(* IEC 61131-3 sources: iec-checker/test/st, 29 files *)

(* ---- declaration-analysis.st ---- *)
(* This demo includes some declaration errors *)
TYPE
    (* String types *)
    ST0 : STRING[5];                               (* OK *)
    ST1 : STRING;                                  (* OK *)
    ST2 : STRING[5] := 'foo';                      (* OK *)
    ST3 : STRING := 'platform_dependent';          (* OK *)
    ST4 : STRING[5] := "foobar";                   (* Error *)

    (* Subrange types *)
    ANALOG_DATA1 : INT (-4095 .. 4095);          (* OK *)
    ANALOG_DATA1 : INT (-4095 .. 4095) := 2000;  (* OK *)
    ANALOG_DATA1 : INT (-4095 .. 4095) := 4095;  (* OK: See 6.4.4.4.1 *)
    ANALOG_DATA1 : INT (-4095 .. 4095) := -4095; (* OK: See 6.4.4.4.1 *)
    ANALOG_DATA2 : INT (-4095 .. 4095) := 4099;  (* Error *)
    ANALOG_DATA2 : INT (-4095 .. 4095) := -4096; (* Error *)
END_TYPE

(* ---- merge-1.st ---- *)
TYPE example_struct :
  STRUCT
    Field : BOOL;
  END_STRUCT
END_TYPE

(* ---- plcopen-cp13.st ---- *)
(* Uncompatible: Recursive functions are forbidden *)
FUNCTION Factorial : INT
    VAR_INPUT
        X : INT;
    END_VAR

    IF X > 1 THEN
        Factorial := Factorial(X - 1) * X;
    ELSE
        Factorial := X;
    END_IF;
END_FUNCTION

(* Compatible iterative implementation *)
FUNCTION Factorial_good : INT
    VAR_INPUT
        X : INT;
    END_VAR
    VAR
        Acc : INT;
    END_VAR

    FOR I := 0 TO 100 DO
        Acc := Acc * X;
    END_FOR;
    Factorial := Acc;
END_FUNCTION

(* ---- plcopen-cp3.st ---- *)
FUNCTION demo : INT
    VAR_INPUT
        x1 : INT := 0;
        x2 : INT; (* PLCOPEN-CP3 *)
        x3 : STRING[5]; (* PLCOPEN-CP3 *)
        x4 : WSTRING[25] := 'spaces_disallowed';
        x5 : ARRAY [1..2, 1..3] OF INT; (* PLCOPEN-CP3 *)
        x6: ARRAY [0..7] OF BOOL := [0,1,1,0,0,1,0,0];
        x7 AT %B0 : INT;
    END_VAR
    x1 := 42;
END_FUNCTION

(* ---- plcopen-cp4.st ---- *)
FUNCTION demo : INT
    VAR_INPUT
        x1 AT %MX40 : INT; (* PLCOPEN-CP4 *)
        x2 AT %MX41 : INT; (* PLCOPEN-CP4 *)
        x3 AT %MX510 : INT;
    END_VAR
    x1 := 42;
END_FUNCTION

(* ---- plcopen-n4.st ---- *)
FUNCTION StartMotor : BOOL
  VAR
    goodVar : INT;
    BadVar  : INT;  (* PLCOPEN-N4 *)
  END_VAR
  StartMotor := TRUE;
END_FUNCTION

FUNCTION start_motor : BOOL    (* PLCOPEN-N4 *)
  start_motor := FALSE;
END_FUNCTION

(* ---- plcopen-n6.st ---- *)
FUNCTION Go : BOOL   (* PLCOPEN-N6 *)
  Go := TRUE;
END_FUNCTION

FUNCTION ReadAndScaleTheTemperatureInput : REAL   (* PLCOPEN-N6 *)
  ReadAndScaleTheTemperatureInput := 0.0;
END_FUNCTION

FUNCTION StartFeeding : BOOL
  StartFeeding := TRUE;
END_FUNCTION

(* ---- plcopen-cp16.st ---- *)
FUNCTION_BLOCK MyFB
  VAR x : INT; END_VAR
  x := 0;
END_FUNCTION_BLOCK

PROGRAM MyProgram
  VAR y : INT; END_VAR
  y := 0;
END_PROGRAM

CONFIGURATION config
  RESOURCE res1 ON PLC
    TASK Fast(INTERVAL := T#10ms, PRIORITY := 1);
    TASK Slow(INTERVAL := T#100ms, PRIORITY := 2);
    PROGRAM inst1 WITH Fast : MyProgram;
    PROGRAM inst2 WITH Slow : MyFB;
    PROGRAM inst3 : MyProgram;
  END_RESOURCE
END_CONFIGURATION

(* ---- plcopen-cp17.st ---- *)
FUNCTION_BLOCK FB_CP17_Test
VAR_INPUT
    in_ok_read_only       : INT;   // Compliant: read at least once, never written
    in_violate_unused     : INT;   // Violation: never read
    in_violate_write_only : INT;   // Violation: written, not read
    in_violate_read_write : INT;   // Violation: read but also written

    idx_read_only           : INT;   // Compliant: only read as array index
    idx_violate_write_only  : INT;   // Violation: written, not read
    func_violate_unused     : INT;   // Violation: never use
    func_read_only          : INT;   // Compliant: only read in func call
    func_violate_write      : INT;   // Violation: written in func call
END_VAR

VAR_OUTPUT
    out_ok_written        : INT;   // Compliant: written at least once
    out_violate_unused    : INT;   // Violation: never written
    out_violate_read_only : INT;   // Violation: read but not written
END_VAR

VAR_IN_OUT
    io_ok_read_only       : INT;   // Compliant: read only
    io_ok_write_only      : INT;   // Compliant: written only
    io_ok_read_write      : INT;   // Compliant: both read and written
    io_violate_unused     : INT;   // Violation: neither read nor written
END_VAR

VAR
    temp : INT;
    arr  : ARRAY[0..9] OF INT;
    func : MYFUNC;
END_VAR

(* ===== VAR_INPUT tests ===== *)

(* Compliant: input parameter is read *)
temp := in_ok_read_only + 1;

(* Violation: in_violate_unused is never used *)

(* Violation: input parameter is written *)
in_violate_write_only := 100;

(* Violation: input parameter is both read and written *)
temp := in_violate_read_write;
in_violate_read_write := temp + 1;

(* ===== VAR_OUTPUT tests ===== *)

(* Compliant: output parameter is written *)
out_ok_written := temp;

(* Violation: out_violate_unused is never written *)

(* Violation: output parameter is read but not written *)
temp := out_violate_read_only;

(* ===== VAR_IN_OUT tests ===== *)

(* Compliant: read only *)
temp := temp + io_ok_read_only;

(* Compliant: written only *)
io_ok_write_only := 10;

(* Compliant: both read and written *)
io_ok_read_write := io_ok_read_write + 1;

(* Violation: io_violate_unused is never used *)

(* ===== special tests for LHS handling ===== *)

(* Important case:
   idx_read_only is used only to locate the write target arr[idx_read_only].
   It should be counted as READ, not WRITE.
   However, *)
arr[idx_read_only] := 5;

(* Violation:
   idx_violate_write_only is written, but never read. *)
idx_violate_write_only := 3;

(* Function Call *)
func(func_violate_unused := func_read_only, func_violate_unused => func_violate_write);

END_FUNCTION_BLOCK

(*
 * The reported result should be:
 * 1. in_violate_unused => should be read
 * 2. in_violate_write_only => should not be written, should be read (2 * warnings reported)
 * 3. in_violate_read_write => should not be written
 * 4. out_violate_unused => should be written
 * 5. out_violate_read_only => should be written
 * 6. io_violate_unused => should be written/read
 * 7. idx_violate_write_only => should not be written, should be read (2 * warnings reported)
 * 8. func_violate_unused => never used, should be read
 * 9. func_violate_write => should not be written, should be read (2 * warnings reported)
*)

(* ---- plcopen-cp6.st ---- *)
FUNCTION demo : INT
    VAR_EXTERNAL
        x1 : INT; (* PLCOPEN-CP6 *)
    END_VAR
    x1 := 42;
END_FUNCTION

FUNCTION_BLOCK demo
    VAR_EXTERNAL
        x1 : INT; (* PLCOPEN-CP6 *)
    END_VAR
    x1 := 42;
END_FUNCTION_BLOCK

PROGRAM demo
    VAR_EXTERNAL
        x1 : INT;
    END_VAR
    x1 := 42;
END_PROGRAM

CLASS test1
  VAR_EXTERNAL
    x1 : INT;
  END_VAR

  METHOD PRIVATE count
    x1 := 42;
  END_METHOD

END_CLASS

(* ---- plcopen-cp9.st ---- *)
(* Example from PLCOpen guidelines, page 60.

   The following Function block CHARCURVE has:
   Number of Statements 18
   McCabe complexity of 12
   Prater complexity of 3,89
   Halstead complexity of 44,9
   Elshof complexity of 0,14

  NOTE: I'm not sure how they evaluated number of statements and appropriate
  complexity metrics. I have 4 additional statements for this program, and it
  seems correct for me.
 *)

FUNCTION_BLOCK CHARCURVE
  VAR_INPUT
    IN:INT;
    N:BYTE;
  END_VAR
  (* VAR_IN_OUT *)
    (* P : ARRAY [0 .. 10] OF POINT; *)
  (* END_VAR *)
  VAR_OUTPUT
    OUT:INT;
    ERR: BYTE;
  END_VAR
  VAR
    I:INT;
  END_VAR

  IF N > 1 AND N < 12 THEN
    ERR:=0;
    (* IF IN < P[0].X THEN *)
    IF IN < a THEN
      ERR := 2;
      OUT := DINT_TO_INT(a);
    (* ELSIF IN > P[N-1].X THEN *)
    ELSIF IN > a THEN
      ERR := 2;
      OUT := DINT_TO_INT(a);
    ELSE
      FOR I:=1 TO N-1 DO
        (* IF P[I-1].X >= P[I].X THEN *)
        IF a >= a THEN
          ERR:=1;
          EXIT;
        END_IF;
        (* IF IN <= P[I].X THEN *)
        IF IN <= a THEN
          EXIT;
        END_IF;
      END_FOR;
      IF ERR = 0 THEN
        (* OUT := DINT_TO_INT(P[I].Y - (P[I].X-IN) * (P[I].Y-P[I-1].Y) / (P[I].X-P[I-1].X)); *)
        OUT := DINT_TO_INT(a - (a - IN) * (a - a) / (a - a));
      ELSE
        OUT:=0;
      END_IF;
    END_IF;
  ELSE
    ERR := 4;
  END_IF;
END_FUNCTION_BLOCK

(* ---- plcopen-n10.st ---- *)
TYPE
  Color : (Red, Green, Blue);   (* PLCOPEN-N10 *)
END_TYPE

TYPE
  E_Direction : (North, South, East, West);
END_TYPE

FUNCTION_BLOCK Motor   (* PLCOPEN-N10 *)
  VAR
    speed : INT;
  END_VAR
  speed := 0;
END_FUNCTION_BLOCK

FUNCTION_BLOCK FB_Pump
  VAR
    flow : REAL;
  END_VAR
  flow := 0.0;
END_FUNCTION_BLOCK

(* ---- plcopen-n5.st ---- *)
PROGRAM prog0
  VAR
    local0 : INT;
  END_VAR
  local0 := 0;
END_PROGRAM

FUNCTION_BLOCK Example
  VAR
    MyCalculation : REAL;   (* PLCOPEN-N5 *)
  END_VAR
  MyCalculation := 0.0;
END_FUNCTION_BLOCK

CONFIGURATION config
  VAR_GLOBAL
    MyCalculation : REAL;
  END_VAR
  TASK task0(INTERVAL := T#20ms, PRIORITY := 0);
  PROGRAM instance0 WITH task0 : prog0;
END_CONFIGURATION

(* ---- plcopen-n9.st ---- *)
PROGRAM prog0
  VAR
    local0 : INT;
  END_VAR
  local0 := 0;
END_PROGRAM

FUNCTION_BLOCK MyCalculation   (* PLCOPEN-N9 *)
  VAR
    value : REAL;
  END_VAR
  value := 0.0;
END_FUNCTION_BLOCK

CONFIGURATION config
  VAR_GLOBAL
    MyCalculation : REAL;   (* PLCOPEN-N9 *)
  END_VAR
  TASK task0(INTERVAL := T#20ms, PRIORITY := 0);
  PROGRAM instance0 WITH task0 : prog0;
END_CONFIGURATION

(* ---- dead-code.st ---- *)
FUNCTION dead_code_after_return : INT
  VAR
    counter : INT := 0;
    some_var : INT;
  END_VAR
  counter := counter + 1;
  counter := 2 + 2;
  RETURN;
  some_var := SQRT(16#42); (* UnreachableCode error *)
  some_var := 16#42; (* No additional warnings *)
  some_var := 19;
END_FUNCTION

PROGRAM dead_code_in_the_loops
VAR a : INT; i : INT; END_VAR
  WHILE i < 10 DO
    IF i = 5 THEN
      i := i + 1;
      EXIT;
      i := 19; (* UnreachableCode error *)
      i := 42; (* No additional warnings *)
      i := 42;
    ELSIF i = 6 THEN
      CONTINUE;
      i := 3; (* UnreachableCode error *)
      i := 44; (* No additional warnings *)
      i := 19;
    END_IF;
    i := i + 2;
  END_WHILE;
  I := 0;
END_PROGRAM

(* ---- merge-2.st ---- *)
PROGRAM Program1
  VAR
    instance AT %MW500 : example_struct;
  END_VAR

  %MW500 := TRUE;
END_PROGRAM

(* ---- plcopen-cp1.st ---- *)
(** PLCOPEN-CP1 – Access to a member shall be by name *)

PROGRAM program0
  VAR
    head AT %B0 : INT;
  END_VAR
  %B0 := 42;
END_PROGRAM

(* ---- plcopen-cp25.st ---- *)
PROGRAM demo
    VAR
        I : INT := 10;
        J : REAL := 0.55;
    END_VAR

  I := J; (* PLCOPEN-CP25 *)
  J := I; (* PLCOPEN-CP25 *)
  I := REAL_TO_INT(J);
  J := INT_TO_REAL(I);
END_PROGRAM

(* ---- plcopen-cp26.st ---- *)
CONFIGURATION config
  VAR_GLOBAL
    SharedCounter : INT;
    ReadOnlyVar : INT;
    MultiWriter : INT;
  END_VAR
  TASK task0(INTERVAL := T#20ms, PRIORITY := 0);
  PROGRAM instance0 WITH task0 : Program1;
END_CONFIGURATION

(* Case 1: SharedCounter written by Program1 and Program2 — violation in Program2 *)
PROGRAM Program1
  VAR_EXTERNAL SharedCounter : INT; END_VAR
  VAR_EXTERNAL ReadOnlyVar : INT; END_VAR
  VAR x : INT; END_VAR
  SharedCounter := SharedCounter + 1;
  x := ReadOnlyVar;
END_PROGRAM

PROGRAM Program2
  VAR_EXTERNAL SharedCounter : INT; END_VAR
  VAR_EXTERNAL ReadOnlyVar : INT; END_VAR
  VAR x : INT; END_VAR
  SharedCounter := 0;
  x := ReadOnlyVar;
END_PROGRAM

(* Case 2: MultiWriter written by Program3 and Program4 — violation in Program4 *)
PROGRAM Program3
  VAR_EXTERNAL MultiWriter : INT; END_VAR
  MultiWriter := 1;
END_PROGRAM

PROGRAM Program4
  VAR_EXTERNAL MultiWriter : INT; END_VAR
  MultiWriter := 2;
END_PROGRAM

(* ---- plcopen-cp28.st ---- *)
PROGRAM demo
    VAR
        x : TIME;
    END_VAR

    IF x = T#100MS THEN (* PLCOPEN CP-28 *)
      x := x + 1;
    END_IF;

    IF x <> T#100MS THEN (* PLCOPEN CP-28 *)
      x := x + 1;
    END_IF;

    IF T#100MS = x THEN (* PLCOPEN CP-28 *)
      x := x + 1;
    END_IF;

    IF T#100MS <> x THEN (* PLCOPEN CP-28 *)
      x := x + 1;
    END_IF;

    IF REAL_TO_INT(x) <> 0 THEN
      x := x + 1;
    END_IF;
END_PROGRAM

(* ---- plcopen-cp8.st ---- *)
PROGRAM demo
    VAR
        x : REAL;
    END_VAR

    IF x = 0.0 THEN (* PLCOPEN CP-8 *)
      x := x + 1;
    END_IF;

    IF x <> 0.0 THEN (* PLCOPEN CP-8 *)
      x := x + 1;
    END_IF;

    IF 0.0 = x THEN (* PLCOPEN CP-8 *)
      x := x + 1;
    END_IF;

    IF 0.0 <> x THEN (* PLCOPEN CP-8 *)
      x := x + 1;
    END_IF;

    IF REAL_TO_INT(x) <> 0 THEN
      x := x + 1;
    END_IF;
END_PROGRAM

(* ---- plcopen-l10.st ---- *)
PROGRAM l10
  VAR
    i : INT := 0;
    j : INT := 0;
    flag : INT := 1;
    counter : INT := 0;
  END_VAR

  FOR i := 0 TO 10 DO
    FOR j := 10 TO 100 BY 2 DO
      IF flag THEN
        EXIT; (* PLCOPEN-CP10 *)
      END_IF;
      counter := counter + 1;
      IF j = 10 THEN
        CONTINUE; (* PLCOPEN-CP10 *)
      END_IF;
      EXIT; (* PLCOPEN-CP10 *)
    END_FOR;
  END_FOR;
END_PROGRAM

(* ---- plcopen-l13.st ---- *)
PROGRAM l13
  VAR
    i : INT := 0;
    j : INT := 0;
    x : INT := 0;
    WORDS : ARRAY[0..100] OF STRING;
    value : STRING := 'val';
  END_VAR

  (* Case 1: Use after FOR — 2 violations *)
  FOR i := 0 TO 100 BY 2 DO
    IF WORDS[i] = 'Key' THEN EXIT; END_IF;
  END_FOR;
  IF i <= 100 THEN
    WORDS[i + 1] := value;
  END_IF;

  (* Case 2: No violation — variable not used after loop *)
  FOR j := 0 TO 10 DO
    x := j;
  END_FOR;

  (* Case 3: Reuse as control var in subsequent FOR — no violation *)
  FOR i := 0 TO 10 DO
    x := i;
  END_FOR;
  FOR i := 0 TO 20 DO
    x := i;
  END_FOR;

  (* Case 4: Nested FOR — outer var used after inner loop — violation *)
  FOR i := 0 TO 10 DO
    FOR j := 0 TO 5 DO
      x := j;
    END_FOR;
    x := j;
  END_FOR;

  (* Case 5: Use in expression after FOR — violation *)
  FOR j := 0 TO 10 DO
    x := j;
  END_FOR;
  x := j + 1;
END_PROGRAM

(* ---- plcopen-l17.st ---- *)
(** PLCOPEN-L17 – Each IF instruction should have an ELSE clause

    Reference: PLCopen Coding Guidelines 6.5.9. *)

PROGRAM program0
  VAR
    a : INT;
  END_VAR

  IF (a = 42) (* PLCOPEN-L17 *)
    THEN
      a := 0;
  END_IF;

  IF (a = 42) (* no warning *)
    THEN
      a := 0;
    ELSE
      a := 19;
  END_IF;

END_PROGRAM

(* ---- plcopen-l22.st ---- *)
PROGRAM l22
  VAR
    i : INT := 0;
    j : INT := 0;
    arr : ARRAY[0..10] OF INT;
  END_VAR

  (* Case 1: Direct assignment in body — violation *)
  FOR i := 0 TO 10 BY 2 DO
    IF arr[i] = 42 THEN
      i := 10;
    END_IF;
  END_FOR;

  (* Case 2: No violation — different variable *)
  FOR i := 0 TO 10 DO
    j := i + 1;
  END_FOR;

  (* Case 3: Nested FOR — inner loop modifies outer var — violation *)
  FOR i := 0 TO 10 DO
    FOR j := 0 TO 5 DO
      i := j;
    END_FOR;
  END_FOR;

  (* Case 4: Nested FOR — inner loop modifies its own var — violation *)
  FOR i := 0 TO 10 DO
    FOR j := 0 TO 5 DO
      j := 0;
    END_FOR;
  END_FOR;
END_PROGRAM

(* ---- plcopen-n1.st ---- *)
PROGRAM l10
  VAR
    a AT %MW10.2.4.1 : INT;
  END_VAR

   %MW10.2.4.1 := 42; (* PLCOPEN-N1 *)
   a := 42; (* ok *)
END_PROGRAM

(* ---- plcopen-n2.st ---- *)
PROGRAM program0
  VAR
    iCounter : INT;
    Counter  : INT;   (* PLCOPEN-N2 *)
    xReady   : BOOL;
    Ready    : BOOL;  (* PLCOPEN-N2 *)
  END_VAR

  iCounter := Counter;
  xReady := Ready;
END_PROGRAM

(* ---- plcopen-n3.st ---- *)
PROGRAM program0
  VAR
    FOR_B : INT; (* PLCOPEN-N3 *)
    NO_FALSE_POSITIVE : INT;
    IF_A : INT; (* PLCOPEN-N3 *)
    TOF : INT; (* PLCOPEN-N3 *)
    OK_ALLOWED : INT;
  END_VAR

  FOR_B := IF_A / 1;
END_PROGRAM

(* ---- plcopen-n8.st ---- *)
PROGRAM program0
  VAR
    CleanName : INT;
    another_clean_name : INT;
  END_VAR
  CleanName := another_clean_name;
END_PROGRAM
